TYPE M2ZAxisStatuses :
STRUCT
	///Is the axis healthy?
	healthStatus: HealthStatus;
END_STRUCT
END_TYPE

(* stored: Version 1.1.0.1, ProductVersion 3.1.4019.2
   DUT M2ZAxisStatuses: Id {3fde5f31-9bae-4082-a091-a58b4d5e5fd7} *)
